(* CoDeSys 2.3 library: SysLibAlarmTrend.lib *)
(* Libraries: TcBase.lib 5.3.04 15:32:36, TcUtilities.lib 25.8.05 11:28:52, TcSystem.lib 7.6.04 13:34:04, Standard.LIB 5.6.98 09:45:02 *)

(* Global variable list: Globale_Variablen *)
VAR_GLOBAL CONSTANT
	SORT_ASCENDING : DWORD := 16#80000000;
	SORT_DESCENDING: DWORD := 16#00000000;
	SORT_NORMALDATE: DWORD := 16#00000001;	(* atm only one date is used *)
	SORT_PRIORITY: DWORD := 16#00000002;	(* sort by priority *)
	SORT_STATE: DWORD := 16#00000004; (* sort by alarmstate *)
	SORT_ALARMCLASS : DWORD := 16#00000008; (* sort by AlarmClassName (String) *)
	ST_INTERNDATEFORMAT : STRING := 'dd.MM.yyyy';
	ST_INTERNTIMEFORMAT : STRING := 'hh:mm:ss';
END_VAR
VAR_GLOBAL
	STAlarmTrend_Text:STRING(255);
	STAlarmTime_TempVar:STAlarmTime;
	STAlarmTime_TempVarCycle:TIME;
	STAlarmTime_TempVarLastCycle:TIME;
	dwTempSize: DWORD;

	sysTime : SysTime64;
	sysTimeStruct : SystemTimeDate;

END_VAR

(* Data type *)
TYPE FILETIME :
STRUCT
	dtCreation:DT;
	dtLastAccess:DT;
	dtLastModification:DT;
END_STRUCT
END_TYPE

(* Data type *)
TYPE STAlarm :
STRUCT
	nID: INT;
	bDeactivation : BOOL;
	dDeadband : REAL;
	dLimit : REAL;
	dTargetValue : REAL;
	dValue : REAL;
	atDate : STAlarmTime;
	btPriority : BYTE;
	btState : BYTE;
	stMessage : STRING (255);
	stType : STRING (10);
	btType : BYTE;
	stExpression : STRING (255);
	stLimit : STRING;
	stDeadband : STRING;
	stTargetValue : STRING;
	pAlarmClass : POINTER TO STAlarmClass;
	bIsSelected : BOOL;
	bToAcknowledge : BOOL;
	btEvent : BYTE;
	stClassName :STRING;
	bHistoryAlarm : BOOL;
END_STRUCT
END_TYPE

(* Data type *)
TYPE STAlarmClass :
STRUCT
	stName : STRING;
	iID : INT;
	arrBGColors: ARRAY [0..2] OF DWORD;
	arrFGColors: ARRAY [0..2] OF DWORD;
	arrBitmaps: ARRAY [0..2] OF INT;
	btAckType : BYTE;
END_STRUCT
END_TYPE

(* Data type *)
TYPE STAlarmGroup :
STRUCT
	stPath : STRING;
	iAlarmCount : INT;
	arrAlarms : ARRAY [0..50] OF POINTER TO STAlarm;
END_STRUCT
END_TYPE

(* Data type *)
TYPE STAlarmTime :
STRUCT
	dwTime : TIME;
	dwDate :DATE;
END_STRUCT
END_TYPE

(* Data type *)
TYPE STDatabase :
STRUCT
	stFileName:STRING;
	stFileExtension:STRING(3);
	dwMaxRecords:DWORD;
	dwActualRecords:DWORD;
	pdwFileIndex:POINTER TO DWORD;
	pbTrigger:POINTER TO BOOL;
	dwLastFileIndex: DWORD;
	dwLastIndex:DWORD;
	atLastChangeTime : STAlarmTime;
	btFileChangeMode : BYTE;
	dwFileDeleteHours : DWORD;
END_STRUCT
END_TYPE

(* Data type *)
TYPE STTrend :
STRUCT
	rValue:REAL;
	dwTime:TIME;
	dwDate:DATE;
END_STRUCT
END_TYPE

(* Data type *)
TYPE SystemTimeDate :
STRUCT
	dwLowMSecs : DWORD;
	dwHighMsec : DWORD;
   	Year : UINT;
	Month : UINT;
	Day : UINT;
	Hour : UINT;
	Minute : UINT;
	Second : UINT;
	Milliseconds : UINT;
	DayOfWeek : UINT;
END_STRUCT
END_TYPE

(* Data type *)
TYPE SysTime64 :
STRUCT
	ulLow:DWORD;
	ulHigh:DWORD;
END_STRUCT
END_TYPE

(* POU AlarmSwap, ST *)
FUNCTION_BLOCK AlarmSwap
VAR_INPUT
	pAlarm1: POINTER TO POINTER TO STAlarm;
	pAlarm2: POINTER TO POINTER TO STAlarm;
END_VAR
VAR_OUTPUT
END_VAR
VAR
	pTemp: POINTER TO STAlarm;
END_VAR
pTemp  := pAlarm1^;
pAlarm1^ := pAlarm2^;
pAlarm2^ := pTemp;
END_FUNCTION_BLOCK

(* POU ChangeAlarmState, ST *)
FUNCTION ChangeAlarmState : BOOL
VAR_INPUT
	pAlarm : POINTER TO STAlarm;
	iEvent : DWORD;
END_VAR
VAR
	btAck : BYTE;
	bDoAction : BOOL := FALSE;
END_VAR
btAck := pAlarm^.pAlarmClass^.btAckType;
IF (iEvent = 2) THEN
	(* reset toAck Flag *)
	pAlarm^.bToAcknowledge := FALSE;
END_IF
pAlarm^.btEvent := DWORD_TO_BYTE (iEvent);
CASE pAlarm^.btState OF
	0:
		IF (iEvent = 1) THEN
			pAlarm^.btState := 1;
			bDoAction := TRUE;
		END_IF
	1:
		IF (iEvent = 4 AND btAck  = 0) THEN
			pAlarm^.btState := 0;
			bDoAction := TRUE;
		ELSIF (iEvent = 4 AND (btAck = 1 OR btAck = 3)) THEN
			pAlarm^.btState := 4;
			bDoAction := TRUE;
		ELSIF (iEvent = 2 AND (btAck = 1 OR btAck = 3)) THEN
			pAlarm^.btState := 2;
			bDoAction := TRUE;
		END_IF
	2:
		IF (iEvent = 4 AND btAck = 1) THEN
			pAlarm^.btState := 0;
			bDoAction := TRUE;
		ELSIF (iEvent = 4 AND (btAck = 2 OR btAck = 3)) THEN
			bDoAction := TRUE;
			pAlarm^.btState := 4;
		END_IF
	4:
		IF (iEvent = 2) THEN
			bDoAction := TRUE;
			pAlarm^.btState := 0;
		ELSIF (iEvent = 1) THEN
			bDoAction := TRUE;
			pAlarm^.btState := 1;
		END_IF;
END_CASE
ChangeAlarmState := bDoAction;
(*
	0 = NORM
	1 = INTO
	2 = ACK
	4 = OUTOF
	0 = NOACK
	1 = ACKINTO
	2 = ACKOUTOF
	3 = ACKALL
*)
END_FUNCTION

(* POU ChangeDateTime, ST *)
FUNCTION ChangeDateTime : INT
VAR_INPUT
	pstATime : POINTER TO STAlarmTime;
	iStep:INT;
END_VAR
VAR
	nDays: DWORD;
END_VAR
IF iStep > 0 THEN
	IF TIME_TO_DWORD (pstATime^.dwTime) + iStep > 86400000 THEN
		(* we also have to increment the date *)
		pstATime^.dwTime := DWORD_TO_TIME (TIME_TO_DWORD (pstATime^.dwTime) + iStep - 86400000);
		pstATime^.dwDate := DWORD_TO_DATE (DATE_TO_DWORD (pstATime^.dwDate) + 86400);
	ELSE
		pstATime^.dwTime := DWORD_TO_TIME (TIME_TO_DWORD (pstATime^.dwTime) + iStep);
	END_IF
ELSE
	IF TIME_TO_DWORD (pstATime^.dwTime) < -iStep THEN
		(* we also have to reduce the days *)
		pstATime^.dwTime := DWORD_TO_TIME (86400000 + TIME_TO_DWORD (pstATime^.dwTime) + iStep);
		pstATime^.dwDate := DWORD_TO_DATE (DATE_TO_DWORD (pstATime^.dwDate) - 86400);
	ELSE
		pstATime^.dwTime := DWORD_TO_TIME (TIME_TO_DWORD (pstATime^.dwTime) + iStep);
	END_IF
END_IF
END_FUNCTION

(* POU ChangeLOHIStates, ST *)
FUNCTION ChangeLOHIStates : BOOL
VAR_INPUT
	pArr: POINTER TO ARRAY[0..0] OF POINTER  TO STAlarm;
	count : INT;
END_VAR
VAR
	i : INT;
	j : INT;
END_VAR
FOR i := 0 TO count - 1 DO
	IF pArr^[i]^.btType = 2 AND pArr^[i]^.btState = 1 THEN
		(* LOLO AND INTO*)
		FOR j := 0 TO count - 1 DO
			IF pArr^[j]^.btType = 3 THEN
				IF pArr^[j]^.btState = 1 AND pArr^[j]^.stExpression  = pArr^[i]^.stExpression THEN
					IF ChangeAlarmState (pArr^[j], 2) THEN
						parr^[j]^.atDate := GetCurrentTime (0);
					END_IF
				END_IF
			END_IF
		END_FOR
	ELSIF pArr^[i]^.btType = 5 AND pArr^[i]^.btState = 1 THEN
		(* HIHI AND INTO*)
		FOR j := 0 TO count - 1 DO
			IF pArr^[j]^.btType = 4 THEN
				IF pArr^[j]^.btState = 1 AND pArr^[j]^.stExpression = pArr^[i]^.stExpression THEN
					IF ChangeAlarmState (pArr^[j], 2) THEN
						parr^[j]^.atDate := GetCurrentTime (0);
					END_IF
				END_IF
			END_IF
		END_FOR
	END_IF
END_FOR
ChangeLOHIStates := TRUE;
END_FUNCTION

(* POU GetCurrentTime, ST *)
FUNCTION GetCurrentTime : STAlarmTime
VAR_INPUT
	dwDummy : DWORD;
END_VAR
VAR
(*
	sysTime : SysTime64;
	sysTimeStruct : SystemTimeDate;
	getTime : CurTimeEx;
*)	
	dwDate:DWORD;
	nMonth :INT ;
	nDay:INT;
	i:INT;
	DayOfMonthTable:ARRAY[0..11] OF INT:=31,28,31,30,31,30,31,31,30,31,30,31;
	dwDiffYear:DWORD;
	dwDiffYearDiv:DWORD;
	dwDiffYearMod:DWORD;
	dwCount:DWORD;

END_VAR
(* getTime (SystemTime := sysTime, TimeDate := sysTimeStruct); *)
GetCurrentTime.dwTime := DWORD_TO_TIME(sysTimeStruct.Milliseconds + 1000 * sysTimeStruct.Second+ 60000 * sysTimeStruct.Minute + 3600000 * sysTimeStruct.Hour);

dwDiffYear := sysTimeStruct.Year - 1970;
dwDiffYearDiv := dwDiffYear / 4;
dwDiffYearMod := dwDiffYear MOD 4;
nMonth:=sysTimeStruct.Month;
nDay:= sysTimeStruct.Day;

CASE dwDiffYearMod OF
	0:	dwCount := dwDiffYearDiv;
	1:	dwCount := dwDiffYearDiv;
	2:	 IF nMonth < 3 THEN
			dwCount := dwDiffYearDiv;
		ELSE
			dwCount := dwDiffYearDiv + 1;
		END_IF
	3:	dwCount := dwDiffYearDiv + 1;
END_CASE;

dwDate := (dwDiffYear * 365 + dwCount) * 24 * 3600;
FOR i:=0 TO nMonth-2  DO
	dwDate := dwDate + (DayOfMonthTable[i] * 24 * 3600);
END_FOR

dwDate := dwDate + ((nDay-1) * 24 * 3600);
GetCurrentTime.dwDate := DWORD_TO_DATE(dwDate);
END_FUNCTION

(* POU CompareDate, ST *)
FUNCTION CompareDate : SINT
VAR_INPUT
	pstRecord : POINTER TO BYTE;
	dwDate : DATE;
	dwTime : TIME;
END_VAR
VAR
	pstRecordStart : POINTER TO STRING;
	dwRecordDate : DATE;
	dwRecordTime : TIME:=t#0ms;
	iCurPos : INT;
	iFoundTokens : INT;
	iLength : INT;
END_VAR
(* Returns > 0 if RecordDate > dwDate and dwTime
    Returns = 0 if RecordDate = dwDate and dwTime
    Returns < 0 in any other case *)
pstRecordStart := pstRecord;
iLength := LEN(pstRecordStart^);
WHILE pstRecord^ <>  59 AND iCurPos < iLength DO
	iCurPos := iCurPos+1;
	pstRecord := pstRecord+1;
END_WHILE

IF(iCurPos < iLength) THEN
	pstRecord^ := 0;
	dwRecordDate := DWORD_TO_DATE(STRING_TO_DWORD(pstRecordStart^));
	pstRecord^ := 59;
	pstRecord := pstRecord+1;
	pstRecordStart := pstRecord;
	WHILE pstRecord^ <>  59 AND iCurPos < iLength DO
		iCurPos := iCurPos+1;
		pstRecord := pstRecord+1;
	END_WHILE

	IF(iCurPos < iLength) THEN
		pstRecord^ := 0;
		dwRecordTime := DWORD_TO_TIME(STRING_TO_DWORD(pstRecordStart^));
		pstRecord^ := 59;
	END_IF

	IF(dwRecordDate = dwDate AND dwRecordTime > dwTime) THEN
		CompareDate := 1;
	ELSE
		IF(dwRecordDate > dwDate) THEN
			CompareDate := 1;
		ELSE
			IF(dwRecordDate = dwDate AND dwRecordTime = dwTime) THEN
				CompareDate := 0;
			ELSE
				CompareDate := -1;
			END_IF
		END_IF
	END_IF
ELSE
	CompareDate := -1;
END_IF
END_FUNCTION

(* POU CurTimeEx, ST *)
FUNCTION_BLOCK CurTimeEx
VAR_IN_OUT
	SystemTime: SysTime64;
	TimeDate: SystemTimeDate;
END_VAR
VAR_OUTPUT
END_VAR
VAR
	fbGetSystemTime : GETSYSTEMTIME;
	fbGetTime	:	NT_GetTime;
END_VAR
fbGetTime( START := FALSE );

fbGetSystemTime();
SystemTime.ulHigh := fbGetSystemTime.timeHiDW;
SystemTime.ulLow := fbGetSystemTime.timeLoDW;

fbGetTime(
	NETID:= '' ,
	START:= TRUE,
	TMOUT:= T#5s
);

TimeDate.Day := fbGetTime.TIMESTR.wDay;
TimeDate.DayOfWeek := fbGetTime.TIMESTR.wDayOfWeek;
TimeDate.Milliseconds := fbGetTime.TIMESTR.wMilliseconds;
TimeDate.Hour := fbGetTime.TIMESTR.wHour;
TimeDate.Minute := fbGetTime.TIMESTR.wMinute;
TimeDate.Month := fbGetTime.TIMESTR.wMonth;
TimeDate.Second := fbGetTime.TIMESTR.wSecond;
TimeDate.Year := fbGetTime.TIMESTR.wYear;
END_FUNCTION_BLOCK

(* POU FormatDate, ST *)
FUNCTION FormatDate : STRING
VAR_INPUT
	dDate : DATE;
	stFormatType : STRING;
END_VAR
VAR
	stTemp1: STRING;
	stTemp2: STRING;
	stTemp3:STRING;
	dwTime: DWORD;
	i: INT;
	dwTemp: DWORD;
END_VAR
(* TODO: implement behavior of formatstring *)
stTemp2 := stFormatType;
stTemp1 := DATE_TO_STRING(dDate);
i := FIND(stTemp1, '#');
stTemp3 := MID(stTemp1, 4, i+1);
i := FIND(stTemp2, 'yyyy');
IF(i <> 0) THEN
	stTemp2 := REPLACE(stTemp2, stTemp3, 4, i);
ELSE
	i := FIND(stTemp2, 'yy');
	IF(i <> 0) THEN
		stTemp3 := RIGHT(stTemp3, 2);
		stTemp2 := REPLACE(stTemp2, stTemp3, 4, i);
	END_IF
END_IF

i := FIND(stTemp1, '-');
stTemp3 := MID(stTemp1, 2, i+1);
i := FIND(stTemp2, 'MM');
IF(i <> 0) THEN
	stTemp2 := REPLACE(stTemp2, stTemp3, 2, i);
END_IF

stTemp3 := RIGHT(stTemp1, 2);
i := FIND(stTemp2, 'dd');
IF(i <> 0) THEN
	stTemp2 :=REPLACE(stTemp2, stTemp3, 2, i);
END_IF
FormatDate:=stTemp2;
END_FUNCTION

(* POU FormatTime, ST *)
FUNCTION FormatTime : STRING
VAR_INPUT
	tTime : TIME;
	stFormatType : STRING;
END_VAR
VAR
	i: INT;
	dwTime:DWORD;
	dwTemp: DWORD;
	stTemp:STRING;
	stHelp:STRING;
END_VAR
(*hh, ss, mm supported*)
dwTime := TIME_TO_DWORD(tTime);
stTemp := stFormatType;

i := FIND(stTemp, 'ss');
IF(i <> 0) THEN
	dwTemp := ((dwTime / 1000) MOD 60 );
	IF(dwTemp < 10) THEN
		stHelp :=CONCAT('0',DWORD_TO_STRING(dwTemp));
	ELSE
		stHelp := DWORD_TO_STRING(dwTemp);
	END_IF
	stTemp :=  REPLACE(stTemp, stHelp, 2, i);
END_IF

i := FIND(stTemp, 'mm');
IF(i <> 0) THEN
	dwTemp := ((dwTime / 60000) MOD 60 );
	IF(dwTemp < 10) THEN
		stHelp :=CONCAT('0',DWORD_TO_STRING(dwTemp));
	ELSE
		stHelp := DWORD_TO_STRING(dwTemp);
	END_IF
	stTemp := REPLACE(stTemp, stHelp, 2, i);
END_IF

i := FIND(stTemp, 'hh');
IF(i <> 0) THEN
	dwTemp := ((dwTime / 3600000) MOD 12 );
	IF(dwTemp < 10) THEN
		stHelp :=CONCAT('0',DWORD_TO_STRING(dwTemp));
	ELSE
		stHelp := DWORD_TO_STRING(dwTemp);
	END_IF
	stTemp :=  REPLACE(stTemp, stHelp, 2, i);
END_IF

i := FIND(stTemp, 'HH');
IF(i <> 0) THEN
	dwTemp := ((dwTime / 3600000) MOD 24 );
	IF(dwTemp < 10) THEN
		stHelp :=CONCAT('0',DWORD_TO_STRING(dwTemp));
	ELSE
		stHelp := DWORD_TO_STRING(dwTemp);
	END_IF
	stTemp :=  REPLACE(stTemp, stHelp, 2, i);
END_IF

FormatTime:=stTemp;
END_FUNCTION

(* POU GenerateAlarmString, ST *)
FUNCTION GenerateAlarmString : STRING (255)
VAR_INPUT
	pAlarm: POINTER TO STAlarm;
END_VAR
VAR
	stTemp : STRING (255);
END_VAR
stTemp := DWORD_TO_STRING (DATE_TO_DWORD(pAlarm^.atDate.dwDate));
stTemp := CONCAT (stTemp, ';');
stTemp :=  CONCAT (stTemp, DWORD_TO_STRING (TIME_TO_DWORD(pAlarm^.atDate.dwTime)));
stTemp := CONCAT (stTemp, ';');
stTemp := CONCAT (stTemp, FormatDate (pAlarm^.atDate.dwDate, 'dd.MM.yyyy'));
stTemp := CONCAT (stTemp, ';');
stTemp := CONCAT (stTemp, FormatTime (pAlarm^.atDate.dwTime, 'hh:mm:ss'));
stTemp := CONCAT (stTemp, ';');
stTemp := CONCAT (stTemp, GetAlarmStateString (pAlarm^.btEvent));
stTemp := CONCAT (stTemp, ';');
stTemp := CONCAT (stTemp, pAlarm^.stExpression);
stTemp := CONCAT (stTemp, ';');
stTemp := CONCAT (stTemp, pAlarm^.stType);
stTemp := CONCAT (stTemp, ';');
stTemp := CONCAT (stTemp, pAlarm^.stLimit);
stTemp := CONCAT (stTemp, ';');
stTemp := CONCAT (stTemp, pAlarm^.stTargetValue);
stTemp := CONCAT (stTemp, ';');
stTemp := CONCAT (stTemp, pAlarm^.stDeadband);
stTemp := CONCAT (stTemp, ';');
stTemp := CONCAT (stTemp, REAL_TO_STRING (pAlarm^.dValue));
stTemp := CONCAT (stTemp, ';');
stTemp := CONCAT (stTemp, pAlarm^.pAlarmClass^.stName);
stTemp := CONCAT (stTemp, ';');
stTemp := CONCAT (stTemp, BYTE_TO_STRING (pAlarm^.btPriority));
stTemp := CONCAT (stTemp, ';');
stTemp := CONCAT (stTemp, pAlarm^.stMessage);
stTemp := CONCAT (stTemp, ';$r$n');
GenerateAlarmString := stTemp;
END_FUNCTION

(* POU GetAlarmStateString, ST *)
FUNCTION GetAlarmStateString : STRING
VAR_INPUT
	state : INT;
END_VAR
VAR
END_VAR
CASE state OF
	0: GetAlarmStateString := 'NORM';
	1: GetAlarmStateString := 'INTO';
	2: GetAlarmStateString := 'ACK';
	4: GetAlarmStateString := 'OUTOF';
END_CASE
END_FUNCTION

(* POU GetAlarmStateValue, ST *)
FUNCTION GetAlarmStateValue : BYTE
VAR_INPUT
	state : STRING;
END_VAR
VAR
END_VAR
IF state = 'NORM' THEN GetAlarmStateValue := 0;
ELSIF state = 'INTO'  THEN GetAlarmStateValue := 1;
ELSIF state = 'ACK'  THEN GetAlarmStateValue := 2;
ELSIF state = 'OUTOF' THEN GetAlarmStateValue := 4;
END_IF
END_FUNCTION

(* POU GetAverage, ST *)
FUNCTION GetAverage : REAL
VAR_INPUT
	pArr : POINTER TO ARRAY [0..0] OF REAL;
	iSize : INT;
END_VAR
VAR
	dSum : REAL := 0;
	i : INT;
END_VAR
FOR i := 0 TO iSize - 1 DO
	dSum := dSum + pArr^[i];
END_FOR
GetAverage := ABS (dSum / iSize);
END_FUNCTION

(* POU GetIndexFromAlarmState, ST *)
FUNCTION GetIndexFromAlarmState : INT
VAR_INPUT
	AlarmState : INT;
END_VAR
VAR
END_VAR
CASE AlarmState OF
	1: GetIndexFromAlarmState := 0;
	2: GetIndexFromAlarmState := 1;
	4: GetIndexFromAlarmState := 2;
END_CASE
END_FUNCTION

(* POU GetNextStoreString, ST *)
FUNCTION_BLOCK GetNextStoreString
VAR_INPUT
	pData: POINTER TO BYTE;
	iSize : DWORD;
	i: DWORD;
	bBeginReading: BOOL;
END_VAR
VAR_OUTPUT
	StoreString : STRING (255);
END_VAR
VAR
	pTemp : POINTER TO BYTE;
	pSetZero : POINTER TO BYTE;
	btTemp : BYTE;
	pstResult : POINTER TO STRING;
	iCurLen : INT;
	iInd : INT;
	iInd2 : INT;
END_VAR
StoreString := '';
pTemp := pData;
iCurLen := 0;
iInd := 0;
WHILE pTemp^ <>  10 AND i < iSize DO
	iCurLen := iCurLen + 1;
	i := i +1;
	pTemp := pTemp + 1;
END_WHILE
IF i < iSize THEN
	pSetZero := pTemp;
	pSetZero^ := 0;		(* exclude \r\n *)
	pstResult := pData;
END_IF
END_FUNCTION_BLOCK

(* POU GetNextToken, ST *)
FUNCTION_BLOCK GetNextToken
VAR_INPUT
	toParse : STRING (255);
	delim : STRING;
END_VAR
VAR_OUTPUT
	stToken : STRING;
END_VAR
VAR
	iPosition : INT;
	stTemp : STRING (255);
	iEndPos : INT;
END_VAR
stTemp := RIGHT (toParse, LEN(toParse) - iPosition);
iEndPos := FIND (stTemp, delim);
iPosition := iPosition + iEndPos;
IF iEndPos > 1 THEN
	stToken := LEFT (stTemp, iEndPos - 1);
ELSE
	stToken := '';
END_IF
END_FUNCTION_BLOCK

(* POU GetVariableValue, ST *)
FUNCTION GetVariableValue : REAL
VAR_INPUT
	stRecord:STRING;
	nVar:INT;
END_VAR
VAR
	nToken: INT;
	stRight: STRING;
	stLeft: STRING;
	nCount:INT;
END_VAR
nToken := FIND(stRecord, ';');
IF nToken > 0 THEN
	stRight:=RIGHT(stRecord, LEN(stRecord)-nToken);
END_IF

nToken := FIND(stRight, ';');
IF nToken > 0 THEN
	stRight:=RIGHT(stRight, LEN(stRight)-nToken);
END_IF



(*2 ';' contains  *)
FOR nCount := 0 TO nVar DO
	nToken:= FIND(stRight, ';');
	IF(LEN(stRight)-nToken  > 1) THEN
		(* Name of Variable*)
		stLeft:=LEFT(stRight, nToken - 1);

		stRight:=RIGHT(stRight, LEN(stRight)-nToken);
	END_IF

	nToken:= FIND(stRight, ';');
	stLeft:=LEFT(stRight, nToken - 1);
	stRight:=RIGHT(stRight, LEN(stRight)-nToken);
	(* Value of Variable *)
	IF nCount = nVar THEN
		GetVariableValue:=STRING_TO_REAL(stLeft);
	END_IF
END_FOR
END_FUNCTION

(* POU IsIPAddress, ST *)
FUNCTION IsIPAddress : BOOL
VAR_INPUT
	stServer:STRING;
END_VAR
VAR
	iPos : INT;
	stTemp : STRING;
END_VAR
IsIPAddress := FALSE;
iPos := FIND(stServer, '.');
IF iPos > 0 THEN
	stTemp := RIGHT(stServer, LEN(stServer)-iPos);
	iPos := FIND(stTemp, '.');
	IF iPos > 0 THEN
		stTemp := RIGHT(stTemp, LEN(stTemp)-iPos);
		iPos := FIND(stTemp, '.');
		IF iPos > 0 THEN
			IsIPAddress := TRUE;
		END_IF
	END_IF
END_IF
END_FUNCTION

(* POU IsSmallerAlarmTime, ST *)
FUNCTION IsSmallerAlarmTime : BOOL
VAR_INPUT
	time1 : STAlarmTime;
	time2 : STAlarmTime;
END_VAR
VAR
END_VAR
IF (time1.dwDate < time2.dwDate) OR ((time1.dwDate = time2.dwDate) AND (time1.dwTime < time2.dwTime)) THEN
	IsSmallerAlarmTime := TRUE;
ELSE
	IsSmallerAlarmTime := FALSE;
END_IF
END_FUNCTION

(* POU ParseAlarmRecord, ST *)
FUNCTION ParseAlarmRecord : BOOL
VAR_INPUT
	toParse : STRING (255);
	pAlarm : POINTER TO STAlarm;
END_VAR
VAR
	Tokenizer : GetNextToken;
END_VAR
pAlarm^.bDeactivation := FALSE;
pAlarm^.bIsSelected := FALSE;
pAlarm^.bToAcknowledge := FALSE;
pAlarm^.dDeadband := 0;
pAlarm^.dLimit := 0;
pAlarm^.dTargetValue := 0;
pAlarm^.dValue := 0;
pAlarm^.pAlarmClass := 0;
Tokenizer.toParse := toParse;
Tokenizer.delim := ';';
Tokenizer ();
pAlarm^.atDate.dwDate := DWORD_TO_DATE (STRING_TO_DWORD (Tokenizer.stToken));
Tokenizer ();
pAlarm^.atDate.dwTime := DWORD_TO_TIME (STRING_TO_DWORD (Tokenizer.stToken));
Tokenizer ();
Tokenizer ();	(* jump over formated date *)
Tokenizer (); 	(* jump over formated time *)
pAlarm^.btEvent := pAlarm^.btState := GetAlarmStateValue (Tokenizer.stToken);
Tokenizer ();
pAlarm^.stExpression := Tokenizer.stToken;
Tokenizer ();
pAlarm^.stType := Tokenizer.stToken;
Tokenizer ();
pAlarm^.stLimit := Tokenizer.stToken;
Tokenizer ();
pAlarm^.stTargetValue := Tokenizer.stToken;
Tokenizer ();
pAlarm^.stDeadband := Tokenizer.stToken;
Tokenizer ();
pAlarm^.dValue := STRING_TO_REAL (Tokenizer.stToken);
Tokenizer ();
pAlarm^.stClassName := Tokenizer.stToken;
Tokenizer ();
pAlarm^.btPriority := STRING_TO_BYTE (Tokenizer.stToken);
Tokenizer ();
pAlarm^.stMessage := Tokenizer.stToken;
pAlarm^.bHistoryAlarm := TRUE;
END_FUNCTION

(* POU ParseDate, ST *)
FUNCTION ParseDate : DATE
VAR_INPUT
	stDate : STRING;
	stFormat : STRING;
END_VAR
VAR
END_VAR
(* TODO: implement behavior of formatstring *)
ParseDate := STRING_TO_DATE (stDate);
END_FUNCTION

(* POU ParseTime, ST *)
FUNCTION ParseTime : TIME
VAR_INPUT
	stTime:STRING;
	stFormat : STRING;
END_VAR
VAR
END_VAR
(* TODO: implement behavior of formatstring *)
ParseTime := STRING_TO_TIME (stTime);
END_FUNCTION

(* POU ParseTrendRecord, ST *)
FUNCTION ParseTrendRecord : INT
VAR_INPUT
	stRecord:STRING;
	tTime:POINTER TO TIME;
	dDate:POINTER TO DATE;
END_VAR
VAR
	nToken: INT := 1;
	stLeft: STRING;
	stRight: STRING;
	nVars:INT;
END_VAR
nToken := FIND(stRecord, ';');
stLeft:=LEFT(stRecord, nToken - 1);
stRight:=RIGHT(stRecord, LEN(stRecord)-nToken);

dDate^ := DWORD_TO_DATE(STRING_TO_DWORD(stLeft));

nToken := FIND(stRight, ';');
stLeft:=LEFT(stRight, nToken - 1);
stRight:=RIGHT(stRight, LEN(stRight)-nToken);


tTime^ := DWORD_TO_TIME(STRING_TO_DWORD(stLeft));

(*2 ';' contains  *)
WHILE nToken <> 0 DO
	nToken:= FIND(stRight, ';');
	stRight:=RIGHT(stRight, LEN(stRight)-nToken);

	nToken:= FIND(stRight, ';');
	stRight:=RIGHT(stRight, LEN(stRight)-nToken);

	IF nToken <> 0 THEN
		nVars := nVars + 1;
	END_IF
END_WHILE

ParseTrendRecord:=nVars;
END_FUNCTION

(* POU ReplaceAlarmPlaceholders, ST *)
FUNCTION ReplaceAlarmPlaceholders : STRING(255)
VAR_INPUT
	Message : STRING(255);
	Alarm : POINTER TO STAlarm;
END_VAR
VAR
END_VAR
Message := ReplaceString (Message, 'ALLDEFAULT',' DATE;TIME;STATE;EXPRESSION;TYPE;TARGETVALUE;DEADBAND;VALUE;CLASS;PRIORITY;MESSAGE');
Message := ReplaceString (Message, 'DATE', FormatDate (Alarm^.atDate.dwDate, ST_INTERNDATEFORMAT));
Message := ReplaceString (Message, 'TIME', FormatTime (Alarm^.atDate.dwTime, ST_INTERNTIMEFORMAT));
Message := ReplaceString (Message, 'MESSAGE', Alarm^.stMessage);
Message := ReplaceString (Message, 'STATE', GetAlarmStateString (Alarm^.btState));
Message := ReplaceString (Message, 'EXPRESSION', Alarm^.stExpression);
Message := ReplaceString (Message, 'TARGETVALUE', REAL_TO_STRING (Alarm^.dTargetValue));
Message := ReplaceString (Message, 'PRIORITY', BYTE_TO_STRING (Alarm^.btPriority));
Message := ReplaceString (Message, 'TYPE', Alarm^.stType);
Message := ReplaceString (Message, 'CLASS', Alarm^.pAlarmClass^.stName);
Message := ReplaceString (Message, 'VALUE', REAL_TO_STRING (Alarm^.dValue));
Message := ReplaceString (Message, 'DEADBAND', REAL_TO_STRING (Alarm^.dDeadband));
ReplaceAlarmPlaceholders := Message;
END_FUNCTION

(* POU ReplaceString, ST *)
FUNCTION ReplaceString : STRING(255)
VAR_INPUT
	Input : STRING(255);
	ToReplace : STRING(255);
	ReplaceWith : STRING(255);
END_VAR
VAR
	iRepLen : INT;
	iRepStart : INT;
	stTemp : STRING(255);
END_VAR
iRepLen := LEN (ToReplace);
stTemp := Input;
iRepStart := FIND (stTemp, ToReplace);
WHILE iRepStart <> 0 DO
	stTemp := REPLACE (stTemp, ReplaceWith, iRepLen, iRepStart);
	iRepStart := FIND (stTemp, ToReplace);
END_WHILE
ReplaceString := stTemp;
END_FUNCTION

(* POU SortAlarms, ST *)
FUNCTION SortAlarms : BOOL
VAR_INPUT
	pAlarms : POINTER TO ARRAY [0..0] OF POINTER TO STAlarm;
	iCount : INT;
	dwSortInfo : DWORD;
END_VAR
VAR
END_VAR
IF (dwSortInfo AND SORT_NORMALDATE) <> 0 THEN
	SortAlarmsByDate (pAlarms, iCount, dwSortInfo);
ELSIF (dwSortInfo AND (SORT_PRIORITY OR SORT_STATE)) <> 0 THEN
	SortAlarmsByNumber (pAlarms, iCount, dwSortInfo);
ELSIF (dwSortInfo AND SORT_ALARMCLASS) <> 0 THEN
	SortAlarmsByString (pAlarms, iCount, dwSortInfo);
END_IF
END_FUNCTION

(* POU SortAlarmsByDate, ST *)
FUNCTION SortAlarmsByDate : BOOL
VAR_INPUT
	pArr: POINTER TO ARRAY[0..0] OF POINTER  TO STAlarm;
	count : INT;
	flags : DWORD;
END_VAR
VAR
	iSmallest : STAlarmTime;
	iSmallestPos: INT;
	i :INT;
	j: INT;
	asAlarmSwap: AlarmSwap;
	iDir: INT;
	iStart : INT;
	iEnd : INT;
END_VAR
IF (flags AND 16#80000000) <> 0 THEN		(*decide sort direction *)
	iDir := 1;
	iStart := 0;
	iEnd := count - 1;
ELSE
	iDir := -1;
	iStart := count - 1;
	iEnd := 0;
END_IF

(* Sort AlarmArray with SelectionSort *)
FOR i:= iStart TO iEnd BY iDir DO
	iSmallest := pArr^[i]^.atDate;
	iSmallestPos := i;
	FOR j:= i + iDir TO iEnd BY iDir DO
		IF IsSmallerAlarmTime (pArr^[j]^.atDate, iSmallest) THEN
			iSmallest :=pArr^[j]^.atDate;
			iSmallestPos := j;
		END_IF
	END_FOR
	IF NOT (iSmallestPos = i) THEN
		asAlarmSwap (pAlarm1 := ADR(pArr^[i]), pAlarm2 := ADR (pArr^[iSmallestPos]));
	END_IF
END_FOR
END_FUNCTION

(* POU SortAlarmsByNumber, ST *)
FUNCTION SortAlarmsByNumber : BOOL
VAR_INPUT
	pArr: POINTER TO ARRAY[0..0] OF POINTER  TO STAlarm;
	count : INT;
	flags : DWORD;
END_VAR
VAR
	iSmallest : INT;
	iSmallestPos: INT;
	i :INT;
	j: INT;
	asAlarmSwap: AlarmSwap;
	iDir: INT;
	iStart : INT;
	iEnd : INT;
	iVal : INT;
END_VAR
IF (flags AND 16#80000000) <> 0 THEN		(*decide sort direction *)
	iDir := 1;
	iStart := 0;
	iEnd := count - 1;
ELSE
	iDir := -1;
	iStart := count - 1;
	iEnd := 0;
END_IF

(* Sort AlarmArray with SelectionSort *)
FOR i:= iStart TO iEnd BY iDir DO
	IF (flags AND SORT_STATE) <> 0 THEN		(* decide about topical sort_value*)
		iSmallest := pArr^[i]^.btState;
	ELSE
		iSmallest := pArr^[i]^.btPriority;
	END_IF
	iSmallestPos := i;
	FOR j:= i + iDir TO iEnd BY iDir  DO
		IF (flags AND SORT_STATE) <> 0 THEN		(* decide about topical sort_value*)
			iVal := pArr^[j]^.btState;
		ELSE
			iVal := pArr^[j]^.btPriority;
		END_IF
		IF iSmallest > iVal THEN
			iSmallest := iVal;
			iSmallestPos := j;
		END_IF
	END_FOR
	IF NOT (iSmallestPos = i) THEN
		asAlarmSwap (pAlarm1 := ADR(pArr^[i]), pAlarm2 := ADR (pArr^[iSmallestPos]));
	END_IF
END_FOR
END_FUNCTION

(* POU SortAlarmsByString, ST *)
FUNCTION SortAlarmsByString : BOOL
VAR_INPUT
	pArr: POINTER TO ARRAY[0..0] OF POINTER  TO STAlarm;
	count : INT;
	flags : DWORD;END_VAR
VAR
	iSmallest : STRING;
	iSmallestPos: INT;
	i :INT;
	j: INT;
	asAlarmSwap: AlarmSwap;
	iDir: INT;
	iStart : INT;
	iEnd : INT;
END_VAR
IF (flags AND 16#80000000) <> 0 THEN		(*decide sort direction *)
	iDir := 1;
	iStart := 0;
	iEnd := count - 1;
ELSE
	iDir := -1;
	iStart := count - 1;
	iEnd := 0;
END_IF

(* Sort AlarmArray with SelectionSort *)
FOR i:= iStart TO iEnd BY iDir DO
	iSmallest := pArr^[i]^.pAlarmClass^.stName;
	iSmallestPos := i;
	FOR j:= i + iDir TO iEnd BY iDir  DO
		IF iSmallest > pArr^[j]^.pAlarmClass^.stName THEN
			iSmallest := pArr^[j]^.pAlarmClass^.stName ;
			iSmallestPos := j;
		END_IF
	END_FOR
	IF NOT (iSmallestPos = i) THEN
		asAlarmSwap (pAlarm1 := ADR(pArr^[i]), pAlarm2 := ADR (pArr^[iSmallestPos]));
	END_IF
END_FOR
END_FUNCTION
